// TwinCAT 3 PLC project TC3_UnitTest_Learning_Space
// ProgramVersion: 3.1.4024.0
// libraries:
//   Tc2_Standard, * (Beckhoff Automation GmbH)
//   Tc2_System, * (Beckhoff Automation GmbH)
//   Tc3_Module, * (Beckhoff Automation GmbH)
//   Tc3_UnitTest, * (Zerlauth)
// project tree:
//   Classes/ MyCalculatorClass.TcPOU
//   / PlcTask.TcTTO
//   POUs/ MAIN.TcPOU
// (motion and I/O tree: see PLC project tcunit_learning_space)
// real-time tasks:
//   TASK PlcTask: cycle T#10ms, priority 20, ADS port 350
//   TASK PlcTask1: cycle T#10ms, priority 21, ADS port 351
//   TASK PlcTask2: cycle T#10ms, priority 22, ADS port 352

CONFIGURATION TC3_UnitTest_Learning_Space
    RESOURCE PLC ON TwinCAT3
        TASK PlcTask(INTERVAL := T#10ms, PRIORITY := 21);
        PROGRAM MAIN WITH PlcTask : MAIN;
    END_RESOURCE
END_CONFIGURATION

// ---- POUs/MAIN.TcPOU
PROGRAM MAIN
VAR
	fbTestSuites : FB_Testsuites;
	fbTestSuite : FB_Testsuite;
	
	MyCalculator : MyCalculatorClass;
	bExecute: BOOL;
END_VAR

fbTestSuites();
fbTestSuites.M_Add(fbTestSuite);
fbTestSuite();

IF bExecute THEN
	// manual execute | override file path
	fbTestsuites.P_Options.sFilePathName:= 'C:\Test\CalculatorTests.xml';
	bExecute:= NOT fbTestsuites.M_Request(E_Base.Execute);
END_IF

CASE fbTestSuite.P_Testcase OF
	E_Testcase.Start:
		fbTestSuite.P_Assert.M_Equals_INT(2, MyCalculator.Divide(4,2), 'Divide method did not return correct qoutient');
		fbTestSuite.M_Testcase('CalculatorClassShouldDivideTwoValidNumbers',T#1S,'','',1);
			 
	1:
		fbTestSuite.P_Assert.M_Equals_INT(-1, MyCalculator.Divide(4,0), 'Divide METHOD did NOT reject 0 divisor');
		fbTestSuite.M_Testcase('CalculatorClassShouldProhibitADivideByZero',T#1S,'','',E_Testcase.Done);

	E_Testcase.Done:;	 
END_CASE

END_PROGRAM

// ---- Classes/MyCalculatorClass.TcPOU
FUNCTION_BLOCK MyCalculatorClass
VAR
END_VAR

METHOD Divide : INT
VAR_INPUT
	x : INT;
	y : INT;
END_VAR
IF y <> 0 THEN
	Divide := x/y;
ELSE
	Divide := -1;
END_IF
END_METHOD

END_FUNCTION_BLOCK
